// TIA Portal V17 export
// export: Created 2025-07-01T14:25:25.0430709Z, ExportSetting WithDefaults, DisplayName Totally Integrated Automation Portal, DisplayVersion V17 Update 8, DisplayName TIA Portal Openness, DisplayVersion V17 Update 8, DisplayName TIA Portal Version Control Interface, DisplayVersion V17, DisplayName SINAMICS Startdrive Advanced, DisplayVersion V17 SP2, DisplayName SINAMICS Startdrive G110M, G120, G120C, G120D, G120P, G115D, DisplayVersion V17 SP2, DisplayName SINAMICS Startdrive G130, G150, S120, S150, SINAMICS MV, S210, DisplayVersion V17 SP2, DisplayName STEP 7 Professional, DisplayVersion V17 Update 8, DisplayName SINUMERIK ONE STEP 7 Toolbox, DisplayVersion V17 Update 12, DisplayName SINUMERIK ONE PLC Basic Program Plus, DisplayVersion V17 Update 12, DisplayName SINUMERIK 840D sl STEP 7 Toolbox, DisplayVersion V17 Update 12, DisplayName STEP 7 Safety, DisplayVersion V17 Update 6, DisplayName WinCC Advanced, DisplayVersion V17 Update 8
FUNCTION_BLOCK "FB20202_TRUMPF_ACTIVE"   // FB20202, LAD
TITLE = FB20202 ACTIVE TRUMPF
{ S7_Optimized_Access := 'FALSE' }
VERSION : 0.1
// stored: AutoNumber false, IsIECCheckEnabled false, SetENOAutomatically false, UDAEnableTagReadback false
   VAR_INPUT
      iREADY_TO_EMISSION : Bool;
      "AIR COMPRESSED OK" : Bool;
      iPROGRAM_ACTIVE : Bool;
      iExternal_In : Bool;
      iMANUAL_START_REQUEST : Bool;
      iAUTO_START_REQUEST : Bool;
      iMANUAL_STOP_REQUEST : Bool;
      iAUTO_STOP_REQUEST : Bool;
      iProfile_Enable : Bool;
      iStart_Program_Request : Bool;
      iUNIT_RESET_LOCAL_SEQ : Bool;
      iSAFETY_GATES_CLOSED_LOCKED : Bool;
      iPART_PRESENTE : Bool;
      iLASER_READY_SC_STATUS : Bool;
      iMACHINE_ON_DELAYED : Bool;
      iZ_AXIS_IN_POSITION : Bool;
      iUNIT_NO : Int;
   END_VAR
   VAR_OUTPUT
      oEMISSION_SWITCH_ON : Bool;
      oPROGRAM_START : Bool;
      oALARM_PROGRAM_NOT_ACTIVE : Bool;
      oALARM_NO_LASER_EMISSION : Bool;
      oALARM_UNSAFE_STATE : Bool;
      oALARM_UNSAFE_AREA : Bool;
      "oALARM_LASER-DSS_ANALOG_MODE_MISMATCH" : Bool;
      oALARM_Z_AXIS_NOT_IN_POSITION : Bool;
      oSTATION_SEOC_ALARMS : Bool;
   END_VAR
   VAR DB_SPECIFIC
      DATA : "LASER ACTIVE";
      "TIMER FAULT 1" { S7_SetPoint := 'True'} : TON_TIME;
      "TIMER FAULT 2" { S7_SetPoint := 'True'} : TON_TIME;
      "DELAY EXTERNAL IN" { S7_SetPoint := 'True'} : TON_TIME;
   END_VAR
   VAR_TEMP
      DB_NUMBER : DInt;
   END_VAR
   VAR_TEMP   // added for the SCL form of the ladder/FBD networks
      _w1 : Bool;
   END_VAR
BEGIN

NETWORK
TITLE = READ INSTANCE DB NUMBER
      L     DINO;
      +     10#800000;
      T     #DB_NUMBER;

REGION Network 2: STOP GENERAL CONDITIONS
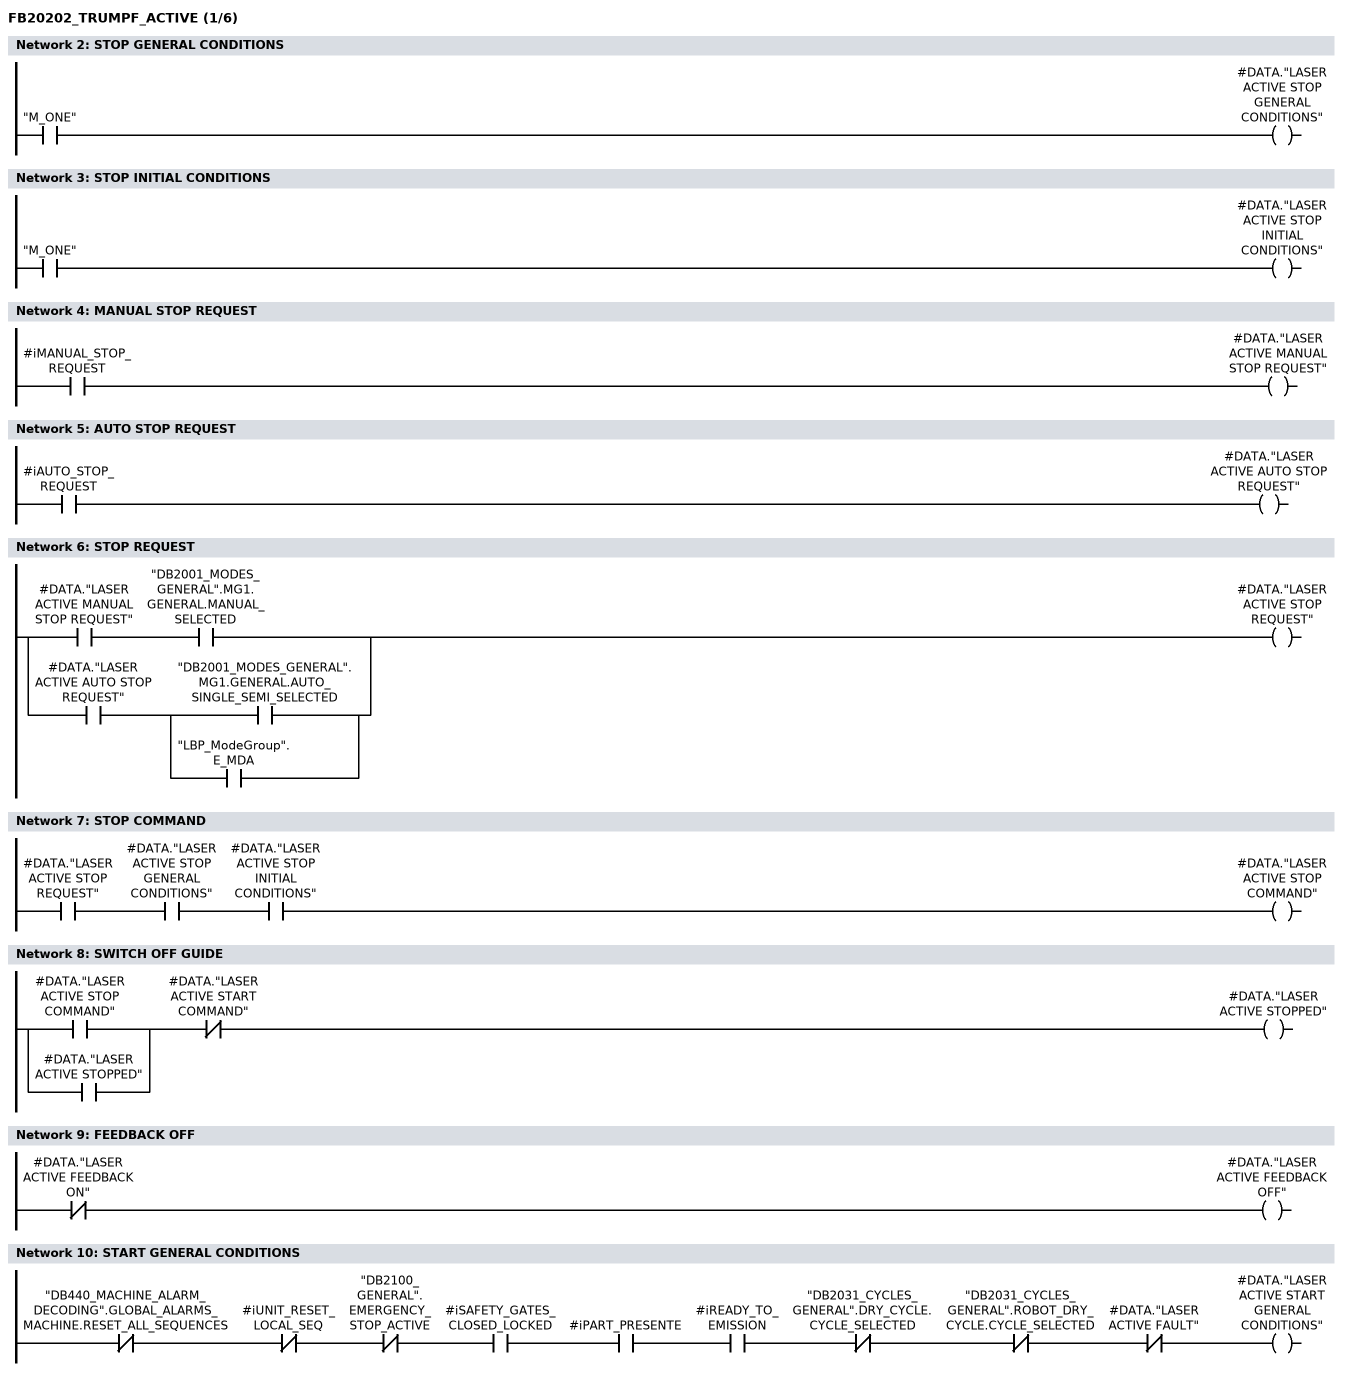
   RUNG wire#powerrail
      Contact( "M_ONE" )
      Coil( #DATA."LASER ACTIVE STOP GENERAL CONDITIONS" )
   END_RUNG
   // the same network as SCL:
   #DATA."LASER ACTIVE STOP GENERAL CONDITIONS" := "M_ONE";
END_REGION

REGION Network 3: STOP INITIAL CONDITIONS
   RUNG wire#powerrail
      Contact( "M_ONE" )
      Coil( #DATA."LASER ACTIVE STOP INITIAL CONDITIONS" )
   END_RUNG
   // the same network as SCL:
   #DATA."LASER ACTIVE STOP INITIAL CONDITIONS" := "M_ONE";
END_REGION

REGION Network 4: MANUAL STOP REQUEST
   RUNG wire#powerrail
      Contact( #iMANUAL_STOP_REQUEST )
      Coil( #DATA."LASER ACTIVE MANUAL STOP REQUEST" )
   END_RUNG
   // the same network as SCL:
   #DATA."LASER ACTIVE MANUAL STOP REQUEST" := #iMANUAL_STOP_REQUEST;
END_REGION

REGION Network 5: AUTO STOP REQUEST
   RUNG wire#powerrail
      Contact( #iAUTO_STOP_REQUEST )
      Coil( #DATA."LASER ACTIVE AUTO STOP REQUEST" )
   END_RUNG
   // the same network as SCL:
   #DATA."LASER ACTIVE AUTO STOP REQUEST" := #iAUTO_STOP_REQUEST;
END_REGION

REGION Network 6: STOP REQUEST
   RUNG wire#powerrail
      Contact( #DATA."LASER ACTIVE MANUAL STOP REQUEST" )
      Contact( "DB2001_MODES_GENERAL".MG1.GENERAL.MANUAL_SELECTED )
      wire#w1
      Coil( #DATA."LASER ACTIVE STOP REQUEST" )
   END_RUNG
   RUNG wire#powerrail
      Contact( #DATA."LASER ACTIVE AUTO STOP REQUEST" )
      wire#w2
      Contact( "DB2001_MODES_GENERAL".MG1.GENERAL.AUTO_SINGLE_SEMI_SELECTED )
   END_RUNG wire#w1
   RUNG wire#w2
      Contact( "LBP_ModeGroup".E_MDA )
   END_RUNG wire#w1
   // the same network as SCL:
   #DATA."LASER ACTIVE STOP REQUEST" := (#DATA."LASER ACTIVE MANUAL STOP REQUEST" AND "DB2001_MODES_GENERAL".MG1.GENERAL.MANUAL_SELECTED) OR (#DATA."LASER ACTIVE AUTO STOP REQUEST" AND ("DB2001_MODES_GENERAL".MG1.GENERAL.AUTO_SINGLE_SEMI_SELECTED OR "LBP_ModeGroup".E_MDA));
END_REGION

REGION Network 7: STOP COMMAND
   RUNG wire#powerrail
      Contact( #DATA."LASER ACTIVE STOP REQUEST" )
      Contact( #DATA."LASER ACTIVE STOP GENERAL CONDITIONS" )
      Contact( #DATA."LASER ACTIVE STOP INITIAL CONDITIONS" )
      Coil( #DATA."LASER ACTIVE STOP COMMAND" )
   END_RUNG
   // the same network as SCL:
   #DATA."LASER ACTIVE STOP COMMAND" := #DATA."LASER ACTIVE STOP REQUEST" AND #DATA."LASER ACTIVE STOP GENERAL CONDITIONS" AND #DATA."LASER ACTIVE STOP INITIAL CONDITIONS";
END_REGION

REGION Network 8: SWITCH OFF GUIDE
   RUNG wire#powerrail
      Contact( #DATA."LASER ACTIVE STOP COMMAND" )
      wire#w1
      I_Contact( #DATA."LASER ACTIVE START COMMAND" )
      Coil( #DATA."LASER ACTIVE STOPPED" )
   END_RUNG
   RUNG wire#powerrail
      Contact( #DATA."LASER ACTIVE STOPPED" )
   END_RUNG wire#w1
   // the same network as SCL:
   #DATA."LASER ACTIVE STOPPED" := (#DATA."LASER ACTIVE STOP COMMAND" OR #DATA."LASER ACTIVE STOPPED") AND NOT #DATA."LASER ACTIVE START COMMAND";
END_REGION

REGION Network 9: FEEDBACK OFF
   RUNG wire#powerrail
      I_Contact( #DATA."LASER ACTIVE FEEDBACK ON" )
      Coil( #DATA."LASER ACTIVE FEEDBACK OFF" )
   END_RUNG
   // the same network as SCL:
   #DATA."LASER ACTIVE FEEDBACK OFF" := NOT #DATA."LASER ACTIVE FEEDBACK ON";
END_REGION

REGION Network 10: START GENERAL CONDITIONS
   RUNG wire#powerrail
      I_Contact( "DB440_MACHINE_ALARM_DECODING".GLOBAL_ALARMS_MACHINE.RESET_ALL_SEQUENCES )
      I_Contact( #iUNIT_RESET_LOCAL_SEQ )
      I_Contact( "DB2100_GENERAL".EMERGENCY_STOP_ACTIVE )
      Contact( #iSAFETY_GATES_CLOSED_LOCKED )
      Contact( #iPART_PRESENTE )
      Contact( #iREADY_TO_EMISSION )
      I_Contact( "DB2031_CYCLES_GENERAL".DRY_CYCLE.CYCLE_SELECTED )
      I_Contact( "DB2031_CYCLES_GENERAL".ROBOT_DRY_CYCLE.CYCLE_SELECTED )
      I_Contact( #DATA."LASER ACTIVE FAULT" )
      Coil( #DATA."LASER ACTIVE START GENERAL CONDITIONS" )
   END_RUNG
   // the same network as SCL:
   #DATA."LASER ACTIVE START GENERAL CONDITIONS" := NOT "DB440_MACHINE_ALARM_DECODING".GLOBAL_ALARMS_MACHINE.RESET_ALL_SEQUENCES AND NOT #iUNIT_RESET_LOCAL_SEQ AND NOT "DB2100_GENERAL".EMERGENCY_STOP_ACTIVE AND #iSAFETY_GATES_CLOSED_LOCKED AND #iPART_PRESENTE AND #iREADY_TO_EMISSION AND NOT "DB2031_CYCLES_GENERAL".DRY_CYCLE.CYCLE_SELECTED AND NOT "DB2031_CYCLES_GENERAL".ROBOT_DRY_CYCLE.CYCLE_SELECTED AND NOT #DATA."LASER ACTIVE FAULT";
END_REGION

REGION Network 11: GENERAL CONDITIONS HELP
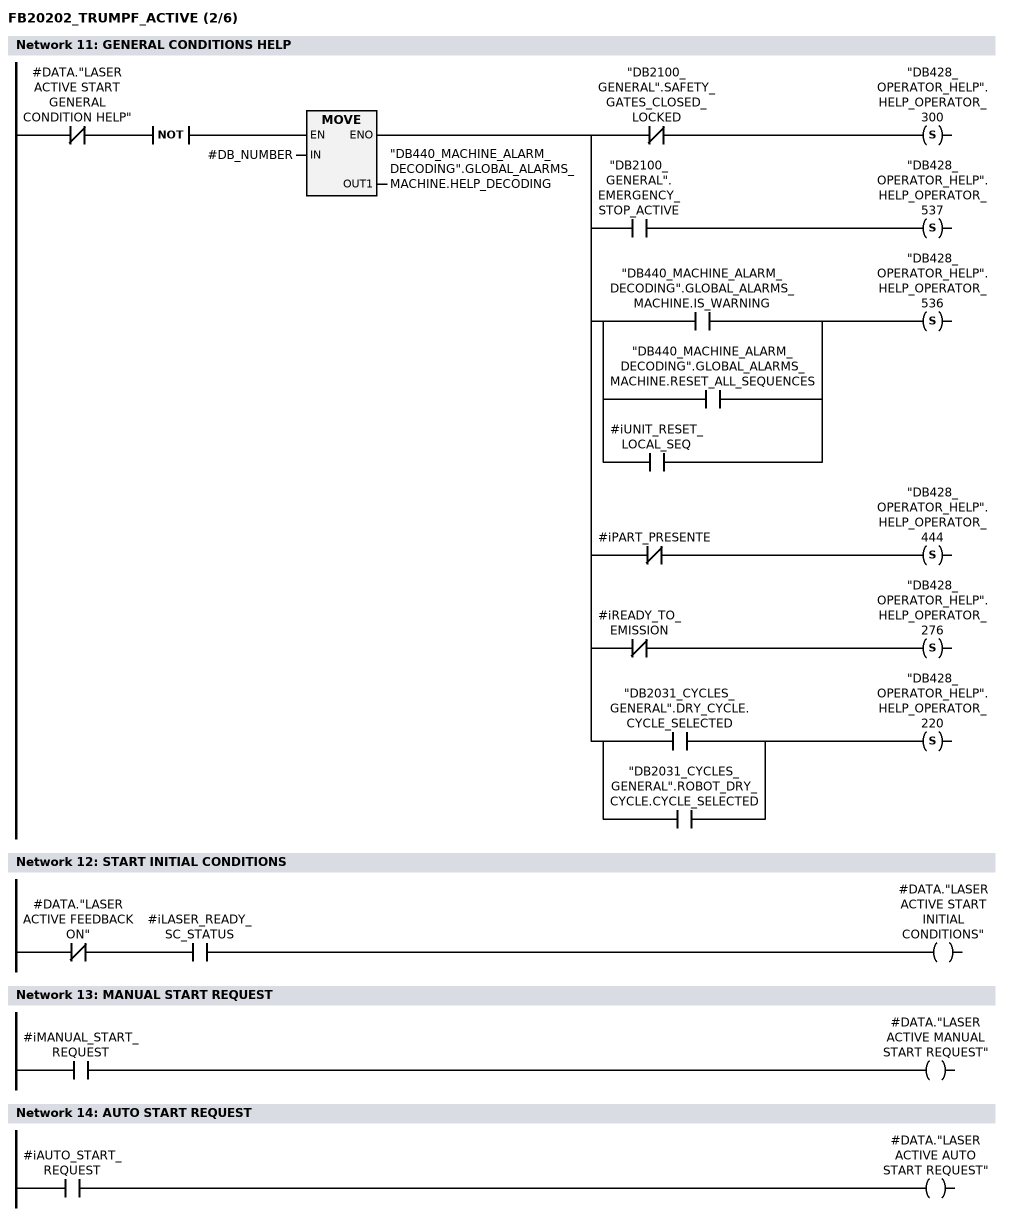
   RUNG wire#powerrail
      I_Contact( #DATA."LASER ACTIVE START GENERAL CONDITION HELP" )
      Not()
      Move(in := #DB_NUMBER, out1 => "DB440_MACHINE_ALARM_DECODING".GLOBAL_ALARMS_MACHINE.HELP_DECODING)
      wire#w1
      I_Contact( "DB2100_GENERAL".SAFETY_GATES_CLOSED_LOCKED )
      S_Coil( "DB428_OPERATOR_HELP".HELP_OPERATOR_300 )
   END_RUNG
   RUNG wire#w1
      Contact( "DB2100_GENERAL".EMERGENCY_STOP_ACTIVE )
      S_Coil( "DB428_OPERATOR_HELP".HELP_OPERATOR_537 )
   END_RUNG
   RUNG wire#w1
      Contact( "DB440_MACHINE_ALARM_DECODING".GLOBAL_ALARMS_MACHINE.IS_WARNING )
      wire#w2
      S_Coil( "DB428_OPERATOR_HELP".HELP_OPERATOR_536 )
   END_RUNG
   RUNG wire#w1
      Contact( "DB440_MACHINE_ALARM_DECODING".GLOBAL_ALARMS_MACHINE.RESET_ALL_SEQUENCES )
   END_RUNG wire#w2
   RUNG wire#w1
      Contact( #iUNIT_RESET_LOCAL_SEQ )
   END_RUNG wire#w2
   RUNG wire#w1
      I_Contact( #iPART_PRESENTE )
      S_Coil( "DB428_OPERATOR_HELP".HELP_OPERATOR_444 )
   END_RUNG
   RUNG wire#w1
      I_Contact( #iREADY_TO_EMISSION )
      S_Coil( "DB428_OPERATOR_HELP".HELP_OPERATOR_276 )
   END_RUNG
   RUNG wire#w1
      Contact( "DB2031_CYCLES_GENERAL".DRY_CYCLE.CYCLE_SELECTED )
      wire#w3
      S_Coil( "DB428_OPERATOR_HELP".HELP_OPERATOR_220 )
   END_RUNG
   RUNG wire#w1
      Contact( "DB2031_CYCLES_GENERAL".ROBOT_DRY_CYCLE.CYCLE_SELECTED )
   END_RUNG wire#w3
   // the same network as SCL:
   #_w1 := NOT (NOT #DATA."LASER ACTIVE START GENERAL CONDITION HELP");
   IF #_w1 THEN "DB440_MACHINE_ALARM_DECODING".GLOBAL_ALARMS_MACHINE.HELP_DECODING := #DB_NUMBER; END_IF;
   IF #_w1 AND NOT "DB2100_GENERAL".SAFETY_GATES_CLOSED_LOCKED THEN
       "DB428_OPERATOR_HELP".HELP_OPERATOR_300 := TRUE;
   END_IF;
   IF #_w1 AND "DB2100_GENERAL".EMERGENCY_STOP_ACTIVE THEN
       "DB428_OPERATOR_HELP".HELP_OPERATOR_537 := TRUE;
   END_IF;
   IF #_w1 AND ("DB440_MACHINE_ALARM_DECODING".GLOBAL_ALARMS_MACHINE.IS_WARNING OR "DB440_MACHINE_ALARM_DECODING".GLOBAL_ALARMS_MACHINE.RESET_ALL_SEQUENCES OR #iUNIT_RESET_LOCAL_SEQ) THEN
       "DB428_OPERATOR_HELP".HELP_OPERATOR_536 := TRUE;
   END_IF;
   IF #_w1 AND NOT #iPART_PRESENTE THEN "DB428_OPERATOR_HELP".HELP_OPERATOR_444 := TRUE; END_IF;
   IF #_w1 AND NOT #iREADY_TO_EMISSION THEN "DB428_OPERATOR_HELP".HELP_OPERATOR_276 := TRUE; END_IF;
   IF #_w1 AND ("DB2031_CYCLES_GENERAL".DRY_CYCLE.CYCLE_SELECTED OR "DB2031_CYCLES_GENERAL".ROBOT_DRY_CYCLE.CYCLE_SELECTED) THEN
       "DB428_OPERATOR_HELP".HELP_OPERATOR_220 := TRUE;
   END_IF;
END_REGION

REGION Network 12: START INITIAL CONDITIONS
   RUNG wire#powerrail
      I_Contact( #DATA."LASER ACTIVE FEEDBACK ON" )
      Contact( #iLASER_READY_SC_STATUS )
      Coil( #DATA."LASER ACTIVE START INITIAL CONDITIONS" )
   END_RUNG
   // the same network as SCL:
   #DATA."LASER ACTIVE START INITIAL CONDITIONS" := NOT #DATA."LASER ACTIVE FEEDBACK ON" AND #iLASER_READY_SC_STATUS;
END_REGION

REGION Network 13: MANUAL START REQUEST
   RUNG wire#powerrail
      Contact( #iMANUAL_START_REQUEST )
      Coil( #DATA."LASER ACTIVE MANUAL START REQUEST" )
   END_RUNG
   // the same network as SCL:
   #DATA."LASER ACTIVE MANUAL START REQUEST" := #iMANUAL_START_REQUEST;
END_REGION

REGION Network 14: AUTO START REQUEST
   RUNG wire#powerrail
      Contact( #iAUTO_START_REQUEST )
      Coil( #DATA."LASER ACTIVE AUTO START REQUEST" )
   END_RUNG
   // the same network as SCL:
   #DATA."LASER ACTIVE AUTO START REQUEST" := #iAUTO_START_REQUEST;
END_REGION

REGION Network 15: START REQUEST
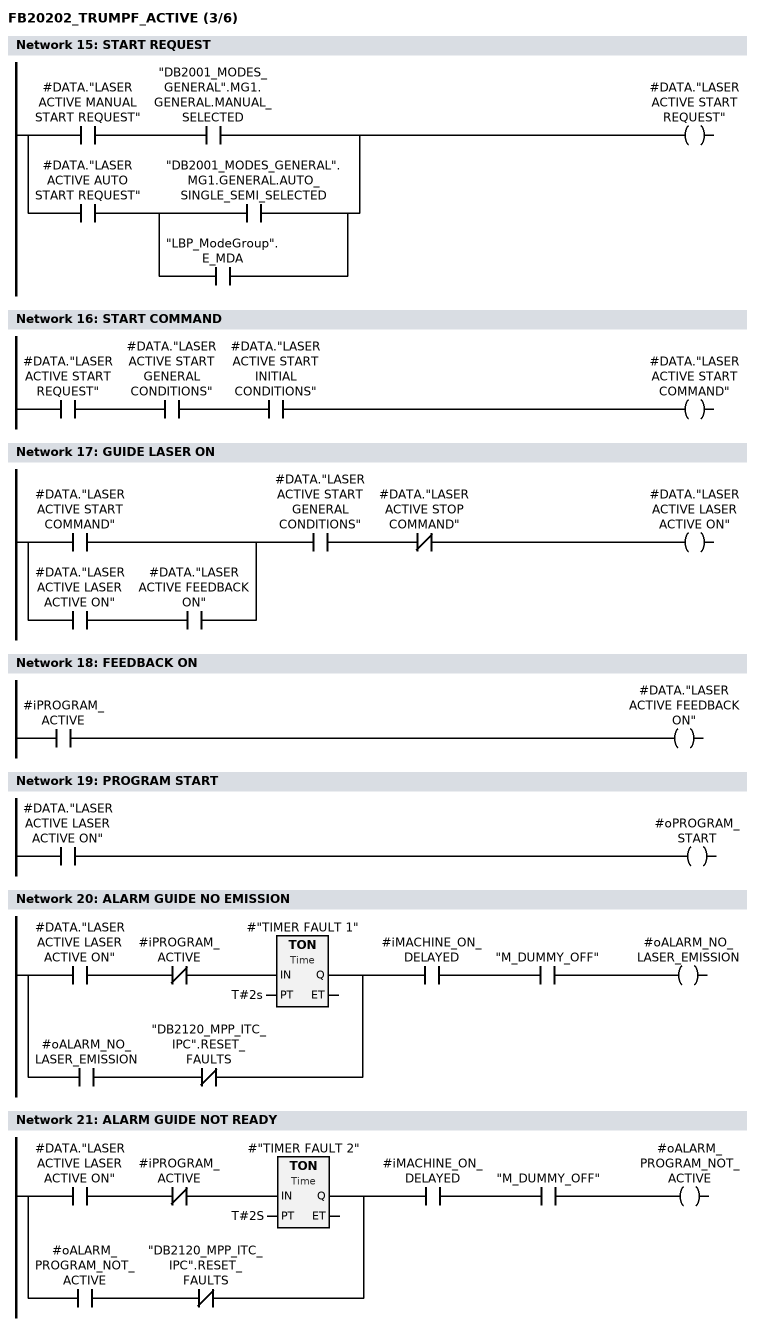
   RUNG wire#powerrail
      Contact( #DATA."LASER ACTIVE MANUAL START REQUEST" )
      Contact( "DB2001_MODES_GENERAL".MG1.GENERAL.MANUAL_SELECTED )
      wire#w1
      Coil( #DATA."LASER ACTIVE START REQUEST" )
   END_RUNG
   RUNG wire#powerrail
      Contact( #DATA."LASER ACTIVE AUTO START REQUEST" )
      wire#w2
      Contact( "DB2001_MODES_GENERAL".MG1.GENERAL.AUTO_SINGLE_SEMI_SELECTED )
   END_RUNG wire#w1
   RUNG wire#w2
      Contact( "LBP_ModeGroup".E_MDA )
   END_RUNG wire#w1
   // the same network as SCL:
   #DATA."LASER ACTIVE START REQUEST" := (#DATA."LASER ACTIVE MANUAL START REQUEST" AND "DB2001_MODES_GENERAL".MG1.GENERAL.MANUAL_SELECTED) OR (#DATA."LASER ACTIVE AUTO START REQUEST" AND ("DB2001_MODES_GENERAL".MG1.GENERAL.AUTO_SINGLE_SEMI_SELECTED OR "LBP_ModeGroup".E_MDA));
END_REGION

REGION Network 16: START COMMAND
   RUNG wire#powerrail
      Contact( #DATA."LASER ACTIVE START REQUEST" )
      Contact( #DATA."LASER ACTIVE START GENERAL CONDITIONS" )
      Contact( #DATA."LASER ACTIVE START INITIAL CONDITIONS" )
      Coil( #DATA."LASER ACTIVE START COMMAND" )
   END_RUNG
   // the same network as SCL:
   #DATA."LASER ACTIVE START COMMAND" := #DATA."LASER ACTIVE START REQUEST" AND #DATA."LASER ACTIVE START GENERAL CONDITIONS" AND #DATA."LASER ACTIVE START INITIAL CONDITIONS";
END_REGION

REGION Network 17: GUIDE LASER ON
   RUNG wire#powerrail
      Contact( #DATA."LASER ACTIVE START COMMAND" )
      wire#w1
      Contact( #DATA."LASER ACTIVE START GENERAL CONDITIONS" )
      I_Contact( #DATA."LASER ACTIVE STOP COMMAND" )
      Coil( #DATA."LASER ACTIVE LASER ACTIVE ON" )
   END_RUNG
   RUNG wire#powerrail
      Contact( #DATA."LASER ACTIVE LASER ACTIVE ON" )
      Contact( #DATA."LASER ACTIVE FEEDBACK ON" )
   END_RUNG wire#w1
   // the same network as SCL:
   #DATA."LASER ACTIVE LASER ACTIVE ON" := (#DATA."LASER ACTIVE START COMMAND" OR (#DATA."LASER ACTIVE LASER ACTIVE ON" AND #DATA."LASER ACTIVE FEEDBACK ON")) AND #DATA."LASER ACTIVE START GENERAL CONDITIONS" AND NOT #DATA."LASER ACTIVE STOP COMMAND";
END_REGION

REGION Network 18: FEEDBACK ON
   RUNG wire#powerrail
      Contact( #iPROGRAM_ACTIVE )
      Coil( #DATA."LASER ACTIVE FEEDBACK ON" )
   END_RUNG
   // the same network as SCL:
   #DATA."LASER ACTIVE FEEDBACK ON" := #iPROGRAM_ACTIVE;
END_REGION

REGION Network 19: PROGRAM START
   RUNG wire#powerrail
      Contact( #DATA."LASER ACTIVE LASER ACTIVE ON" )
      Coil( #oPROGRAM_START )
   END_RUNG
   // the same network as SCL:
   #oPROGRAM_START := #DATA."LASER ACTIVE LASER ACTIVE ON";
END_REGION

REGION Network 20: ALARM GUIDE NO EMISSION
   RUNG wire#powerrail
      Contact( #DATA."LASER ACTIVE LASER ACTIVE ON" )
      I_Contact( #iPROGRAM_ACTIVE )
      { S7_Templates := "time_type := Time" } #"TIMER FAULT 1".TON(pt := T#2s, et =>)
      wire#w1
      Contact( #iMACHINE_ON_DELAYED )
      Contact( "M_DUMMY_OFF" )
      Coil( #oALARM_NO_LASER_EMISSION )
   END_RUNG
   RUNG wire#powerrail
      Contact( #oALARM_NO_LASER_EMISSION )
      I_Contact( "DB2120_MPP_ITC_IPC".RESET_FAULTS )
   END_RUNG wire#w1
   // the same network as SCL:
   #"TIMER FAULT 1"(IN := #DATA."LASER ACTIVE LASER ACTIVE ON" AND NOT #iPROGRAM_ACTIVE, PT := T#2s);   // TON
   #oALARM_NO_LASER_EMISSION := (#"TIMER FAULT 1".Q OR (#oALARM_NO_LASER_EMISSION AND NOT "DB2120_MPP_ITC_IPC".RESET_FAULTS)) AND #iMACHINE_ON_DELAYED AND "M_DUMMY_OFF";
END_REGION

REGION Network 21: ALARM GUIDE NOT READY
   RUNG wire#powerrail
      Contact( #DATA."LASER ACTIVE LASER ACTIVE ON" )
      I_Contact( #iPROGRAM_ACTIVE )
      { S7_Templates := "time_type := Time" } #"TIMER FAULT 2".TON(pt := T#2S, et =>)
      wire#w1
      Contact( #iMACHINE_ON_DELAYED )
      Contact( "M_DUMMY_OFF" )
      Coil( #oALARM_PROGRAM_NOT_ACTIVE )
   END_RUNG
   RUNG wire#powerrail
      Contact( #oALARM_PROGRAM_NOT_ACTIVE )
      I_Contact( "DB2120_MPP_ITC_IPC".RESET_FAULTS )
   END_RUNG wire#w1
   // the same network as SCL:
   #"TIMER FAULT 2"(IN := #DATA."LASER ACTIVE LASER ACTIVE ON" AND NOT #iPROGRAM_ACTIVE, PT := T#2S);   // TON
   #oALARM_PROGRAM_NOT_ACTIVE := (#"TIMER FAULT 2".Q OR (#oALARM_PROGRAM_NOT_ACTIVE AND NOT "DB2120_MPP_ITC_IPC".RESET_FAULTS)) AND #iMACHINE_ON_DELAYED AND "M_DUMMY_OFF";
END_REGION

REGION Network 22: ALARM GUIDE NOT READY
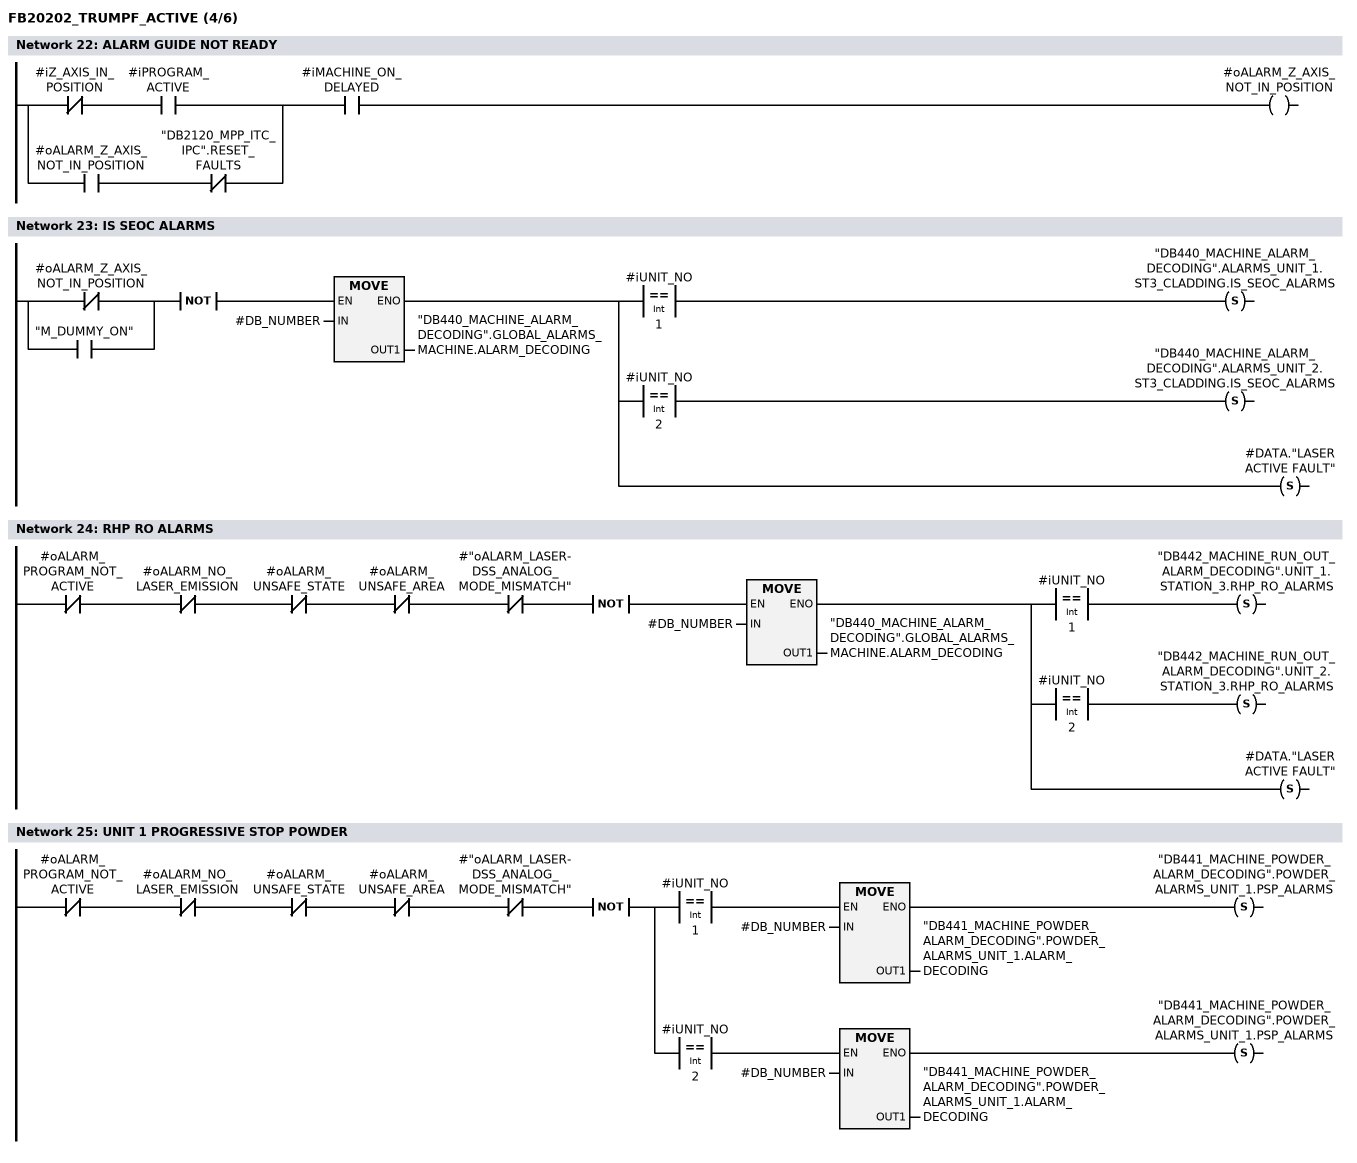
   RUNG wire#powerrail
      I_Contact( #iZ_AXIS_IN_POSITION )
      Contact( #iPROGRAM_ACTIVE )
      wire#w1
      Contact( #iMACHINE_ON_DELAYED )
      Coil( #oALARM_Z_AXIS_NOT_IN_POSITION )
   END_RUNG
   RUNG wire#powerrail
      Contact( #oALARM_Z_AXIS_NOT_IN_POSITION )
      I_Contact( "DB2120_MPP_ITC_IPC".RESET_FAULTS )
   END_RUNG wire#w1
   // the same network as SCL:
   #oALARM_Z_AXIS_NOT_IN_POSITION := ((NOT #iZ_AXIS_IN_POSITION AND #iPROGRAM_ACTIVE) OR (#oALARM_Z_AXIS_NOT_IN_POSITION AND NOT "DB2120_MPP_ITC_IPC".RESET_FAULTS)) AND #iMACHINE_ON_DELAYED;
END_REGION

REGION Network 23: IS SEOC ALARMS
   RUNG wire#powerrail
      I_Contact( #oALARM_Z_AXIS_NOT_IN_POSITION )
      wire#w1
      Not()
      Move(in := #DB_NUMBER, out1 => "DB440_MACHINE_ALARM_DECODING".GLOBAL_ALARMS_MACHINE.ALARM_DECODING)
      wire#w2
      { S7_Templates := "SrcType := Int" } EQ_Contact(in1 := #iUNIT_NO, in2 := 1)
      S_Coil( "DB440_MACHINE_ALARM_DECODING".ALARMS_UNIT_1.ST3_CLADDING.IS_SEOC_ALARMS )
   END_RUNG
   RUNG wire#powerrail
      Contact( "M_DUMMY_ON" )
   END_RUNG wire#w1
   RUNG wire#w2
      { S7_Templates := "SrcType := Int" } EQ_Contact(in1 := #iUNIT_NO, in2 := 2)
      S_Coil( "DB440_MACHINE_ALARM_DECODING".ALARMS_UNIT_2.ST3_CLADDING.IS_SEOC_ALARMS )
   END_RUNG
   RUNG wire#w2
      S_Coil( #DATA."LASER ACTIVE FAULT" )
   END_RUNG
   // the same network as SCL:
   #_w1 := NOT (NOT #oALARM_Z_AXIS_NOT_IN_POSITION OR "M_DUMMY_ON");
   IF #_w1 THEN "DB440_MACHINE_ALARM_DECODING".GLOBAL_ALARMS_MACHINE.ALARM_DECODING := #DB_NUMBER; END_IF;
   IF #_w1 AND (#iUNIT_NO = 1) THEN
       "DB440_MACHINE_ALARM_DECODING".ALARMS_UNIT_1.ST3_CLADDING.IS_SEOC_ALARMS := TRUE;
   END_IF;
   IF #_w1 AND (#iUNIT_NO = 2) THEN
       "DB440_MACHINE_ALARM_DECODING".ALARMS_UNIT_2.ST3_CLADDING.IS_SEOC_ALARMS := TRUE;
   END_IF;
   IF #_w1 THEN #DATA."LASER ACTIVE FAULT" := TRUE; END_IF;
END_REGION

REGION Network 24: RHP RO ALARMS
   RUNG wire#powerrail
      I_Contact( #oALARM_PROGRAM_NOT_ACTIVE )
      I_Contact( #oALARM_NO_LASER_EMISSION )
      I_Contact( #oALARM_UNSAFE_STATE )
      I_Contact( #oALARM_UNSAFE_AREA )
      I_Contact( #"oALARM_LASER-DSS_ANALOG_MODE_MISMATCH" )
      Not()
      Move(in := #DB_NUMBER, out1 => "DB440_MACHINE_ALARM_DECODING".GLOBAL_ALARMS_MACHINE.ALARM_DECODING)
      wire#w1
      { S7_Templates := "SrcType := Int" } EQ_Contact(in1 := #iUNIT_NO, in2 := 1)
      S_Coil( "DB442_MACHINE_RUN_OUT_ALARM_DECODING".UNIT_1.STATION_3.RHP_RO_ALARMS )
   END_RUNG
   RUNG wire#w1
      { S7_Templates := "SrcType := Int" } EQ_Contact(in1 := #iUNIT_NO, in2 := 2)
      S_Coil( "DB442_MACHINE_RUN_OUT_ALARM_DECODING".UNIT_2.STATION_3.RHP_RO_ALARMS )
   END_RUNG
   RUNG wire#w1
      S_Coil( #DATA."LASER ACTIVE FAULT" )
   END_RUNG
   // the same network as SCL:
   #_w1 := NOT (NOT #oALARM_PROGRAM_NOT_ACTIVE AND NOT #oALARM_NO_LASER_EMISSION AND NOT #oALARM_UNSAFE_STATE AND NOT #oALARM_UNSAFE_AREA AND NOT #"oALARM_LASER-DSS_ANALOG_MODE_MISMATCH");
   IF #_w1 THEN "DB440_MACHINE_ALARM_DECODING".GLOBAL_ALARMS_MACHINE.ALARM_DECODING := #DB_NUMBER; END_IF;
   IF #_w1 AND (#iUNIT_NO = 1) THEN
       "DB442_MACHINE_RUN_OUT_ALARM_DECODING".UNIT_1.STATION_3.RHP_RO_ALARMS := TRUE;
   END_IF;
   IF #_w1 AND (#iUNIT_NO = 2) THEN
       "DB442_MACHINE_RUN_OUT_ALARM_DECODING".UNIT_2.STATION_3.RHP_RO_ALARMS := TRUE;
   END_IF;
   IF #_w1 THEN #DATA."LASER ACTIVE FAULT" := TRUE; END_IF;
END_REGION

REGION Network 25: UNIT 1 PROGRESSIVE STOP POWDER
   RUNG wire#powerrail
      I_Contact( #oALARM_PROGRAM_NOT_ACTIVE )
      I_Contact( #oALARM_NO_LASER_EMISSION )
      I_Contact( #oALARM_UNSAFE_STATE )
      I_Contact( #oALARM_UNSAFE_AREA )
      I_Contact( #"oALARM_LASER-DSS_ANALOG_MODE_MISMATCH" )
      Not()
      wire#w1
      { S7_Templates := "SrcType := Int" } EQ_Contact(in1 := #iUNIT_NO, in2 := 1)
      Move(in := #DB_NUMBER, out1 => "DB441_MACHINE_POWDER_ALARM_DECODING".POWDER_ALARMS_UNIT_1.ALARM_DECODING)
      S_Coil( "DB441_MACHINE_POWDER_ALARM_DECODING".POWDER_ALARMS_UNIT_1.PSP_ALARMS )
   END_RUNG
   RUNG wire#w1
      { S7_Templates := "SrcType := Int" } EQ_Contact(in1 := #iUNIT_NO, in2 := 2)
      Move(in := #DB_NUMBER, out1 => "DB441_MACHINE_POWDER_ALARM_DECODING".POWDER_ALARMS_UNIT_1.ALARM_DECODING)
      S_Coil( "DB441_MACHINE_POWDER_ALARM_DECODING".POWDER_ALARMS_UNIT_1.PSP_ALARMS )
   END_RUNG
   // the same network as SCL:
   #_w1 := NOT (NOT #oALARM_PROGRAM_NOT_ACTIVE AND NOT #oALARM_NO_LASER_EMISSION AND NOT #oALARM_UNSAFE_STATE AND NOT #oALARM_UNSAFE_AREA AND NOT #"oALARM_LASER-DSS_ANALOG_MODE_MISMATCH");
   IF #_w1 AND (#iUNIT_NO = 1) THEN
       "DB441_MACHINE_POWDER_ALARM_DECODING".POWDER_ALARMS_UNIT_1.ALARM_DECODING := #DB_NUMBER;
       "DB441_MACHINE_POWDER_ALARM_DECODING".POWDER_ALARMS_UNIT_1.PSP_ALARMS := TRUE;
   END_IF;
   IF #_w1 AND (#iUNIT_NO = 2) THEN
       "DB441_MACHINE_POWDER_ALARM_DECODING".POWDER_ALARMS_UNIT_1.ALARM_DECODING := #DB_NUMBER;
       "DB441_MACHINE_POWDER_ALARM_DECODING".POWDER_ALARMS_UNIT_1.PSP_ALARMS := TRUE;
   END_IF;
END_REGION

REGION Network 26: UNIT 2 MAINTAIN POWDER
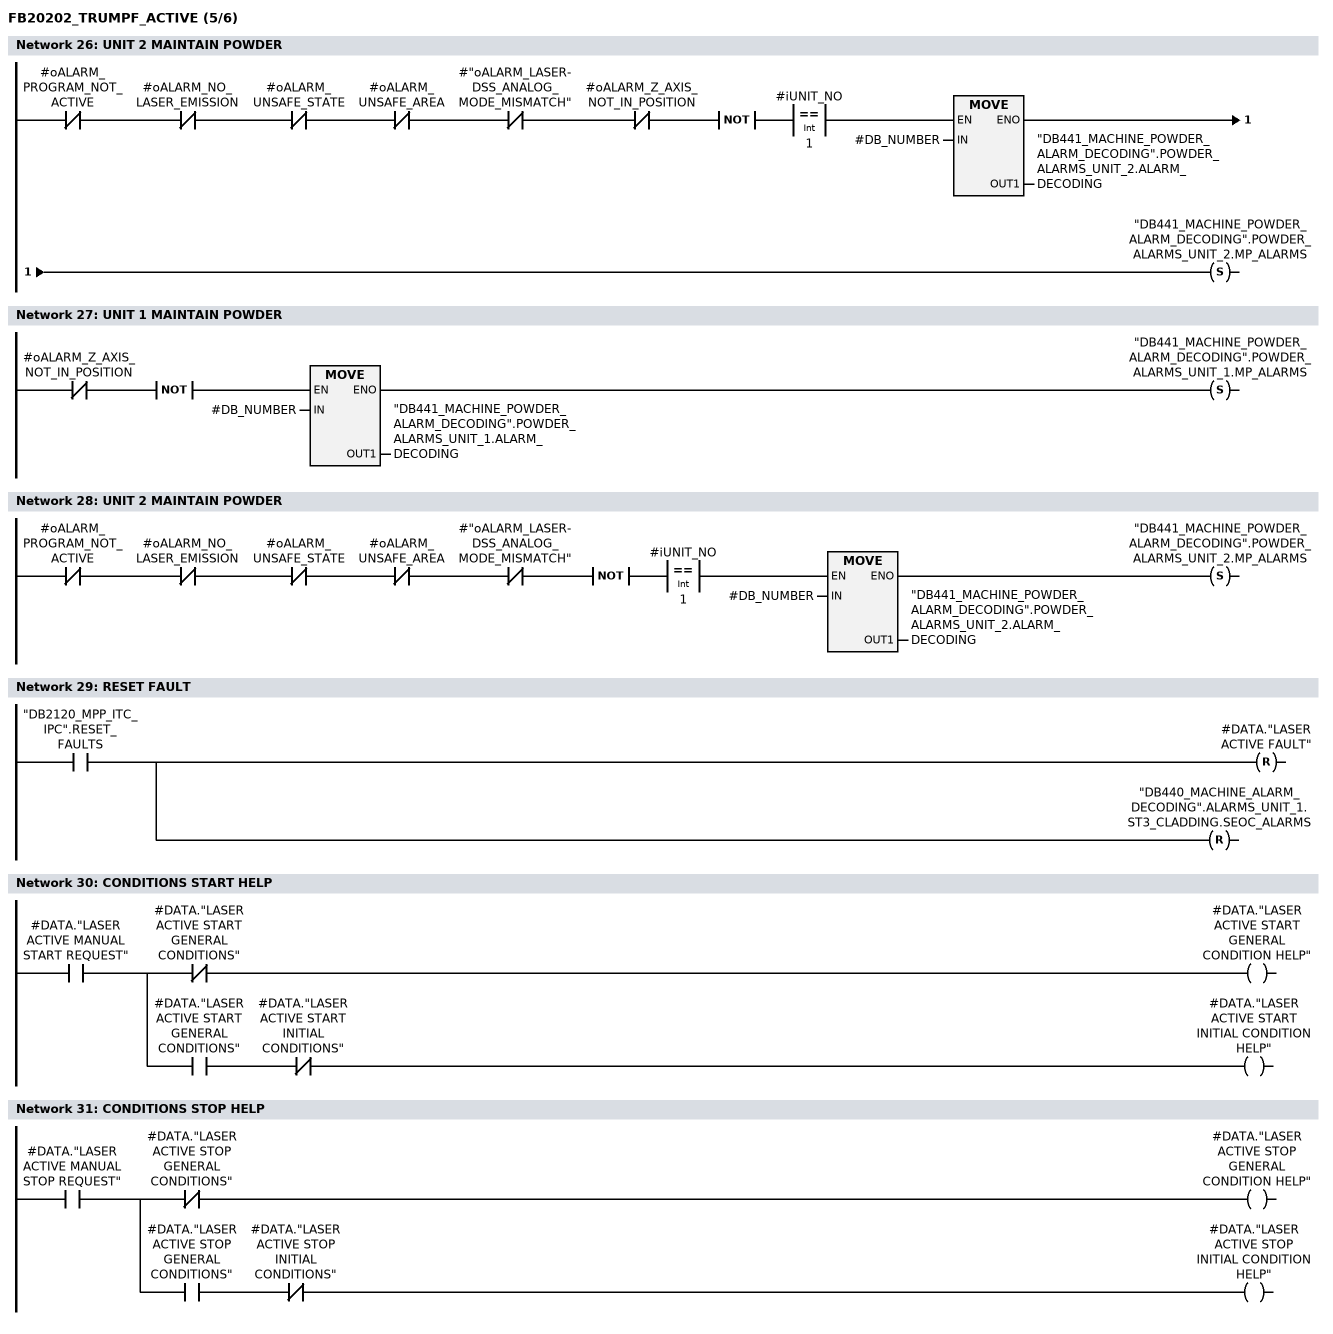
   RUNG wire#powerrail
      I_Contact( #oALARM_PROGRAM_NOT_ACTIVE )
      I_Contact( #oALARM_NO_LASER_EMISSION )
      I_Contact( #oALARM_UNSAFE_STATE )
      I_Contact( #oALARM_UNSAFE_AREA )
      I_Contact( #"oALARM_LASER-DSS_ANALOG_MODE_MISMATCH" )
      I_Contact( #oALARM_Z_AXIS_NOT_IN_POSITION )
      Not()
      { S7_Templates := "SrcType := Int" } EQ_Contact(in1 := #iUNIT_NO, in2 := 1)
      Move(in := #DB_NUMBER, out1 => "DB441_MACHINE_POWDER_ALARM_DECODING".POWDER_ALARMS_UNIT_2.ALARM_DECODING)
      S_Coil( "DB441_MACHINE_POWDER_ALARM_DECODING".POWDER_ALARMS_UNIT_2.MP_ALARMS )
   END_RUNG
   // the same network as SCL:
   IF NOT (NOT #oALARM_PROGRAM_NOT_ACTIVE AND NOT #oALARM_NO_LASER_EMISSION AND NOT #oALARM_UNSAFE_STATE AND NOT #oALARM_UNSAFE_AREA AND NOT #"oALARM_LASER-DSS_ANALOG_MODE_MISMATCH" AND NOT #oALARM_Z_AXIS_NOT_IN_POSITION) AND (#iUNIT_NO = 1) THEN
       "DB441_MACHINE_POWDER_ALARM_DECODING".POWDER_ALARMS_UNIT_2.ALARM_DECODING := #DB_NUMBER;
       "DB441_MACHINE_POWDER_ALARM_DECODING".POWDER_ALARMS_UNIT_2.MP_ALARMS := TRUE;
   END_IF;
END_REGION

REGION Network 27: UNIT 1 MAINTAIN POWDER
   RUNG wire#powerrail
      I_Contact( #oALARM_Z_AXIS_NOT_IN_POSITION )
      Not()
      Move(in := #DB_NUMBER, out1 => "DB441_MACHINE_POWDER_ALARM_DECODING".POWDER_ALARMS_UNIT_1.ALARM_DECODING)
      S_Coil( "DB441_MACHINE_POWDER_ALARM_DECODING".POWDER_ALARMS_UNIT_1.MP_ALARMS )
   END_RUNG
   // the same network as SCL:
   IF NOT (NOT #oALARM_Z_AXIS_NOT_IN_POSITION) THEN
       "DB441_MACHINE_POWDER_ALARM_DECODING".POWDER_ALARMS_UNIT_1.ALARM_DECODING := #DB_NUMBER;
       "DB441_MACHINE_POWDER_ALARM_DECODING".POWDER_ALARMS_UNIT_1.MP_ALARMS := TRUE;
   END_IF;
END_REGION

REGION Network 28: UNIT 2 MAINTAIN POWDER
   RUNG wire#powerrail
      I_Contact( #oALARM_PROGRAM_NOT_ACTIVE )
      I_Contact( #oALARM_NO_LASER_EMISSION )
      I_Contact( #oALARM_UNSAFE_STATE )
      I_Contact( #oALARM_UNSAFE_AREA )
      I_Contact( #"oALARM_LASER-DSS_ANALOG_MODE_MISMATCH" )
      Not()
      { S7_Templates := "SrcType := Int" } EQ_Contact(in1 := #iUNIT_NO, in2 := 1)
      Move(in := #DB_NUMBER, out1 => "DB441_MACHINE_POWDER_ALARM_DECODING".POWDER_ALARMS_UNIT_2.ALARM_DECODING)
      S_Coil( "DB441_MACHINE_POWDER_ALARM_DECODING".POWDER_ALARMS_UNIT_2.MP_ALARMS )
   END_RUNG
   // the same network as SCL:
   IF NOT (NOT #oALARM_PROGRAM_NOT_ACTIVE AND NOT #oALARM_NO_LASER_EMISSION AND NOT #oALARM_UNSAFE_STATE AND NOT #oALARM_UNSAFE_AREA AND NOT #"oALARM_LASER-DSS_ANALOG_MODE_MISMATCH") AND (#iUNIT_NO = 1) THEN
       "DB441_MACHINE_POWDER_ALARM_DECODING".POWDER_ALARMS_UNIT_2.ALARM_DECODING := #DB_NUMBER;
       "DB441_MACHINE_POWDER_ALARM_DECODING".POWDER_ALARMS_UNIT_2.MP_ALARMS := TRUE;
   END_IF;
END_REGION

REGION Network 29: RESET FAULT
   RUNG wire#powerrail
      Contact( "DB2120_MPP_ITC_IPC".RESET_FAULTS )
      wire#w1
      R_Coil( #DATA."LASER ACTIVE FAULT" )
   END_RUNG
   RUNG wire#w1
      R_Coil( "DB440_MACHINE_ALARM_DECODING".ALARMS_UNIT_1.ST3_CLADDING.SEOC_ALARMS )
   END_RUNG
   // the same network as SCL:
   IF "DB2120_MPP_ITC_IPC".RESET_FAULTS THEN
       #DATA."LASER ACTIVE FAULT" := FALSE;
       "DB440_MACHINE_ALARM_DECODING".ALARMS_UNIT_1.ST3_CLADDING.SEOC_ALARMS := FALSE;
   END_IF;
END_REGION

REGION Network 30: CONDITIONS START HELP
   RUNG wire#powerrail
      Contact( #DATA."LASER ACTIVE MANUAL START REQUEST" )
      wire#w1
      I_Contact( #DATA."LASER ACTIVE START GENERAL CONDITIONS" )
      Coil( #DATA."LASER ACTIVE START GENERAL CONDITION HELP" )
   END_RUNG
   RUNG wire#w1
      Contact( #DATA."LASER ACTIVE START GENERAL CONDITIONS" )
      I_Contact( #DATA."LASER ACTIVE START INITIAL CONDITIONS" )
      Coil( #DATA."LASER ACTIVE START INITIAL CONDITION HELP" )
   END_RUNG
   // the same network as SCL:
   #DATA."LASER ACTIVE START GENERAL CONDITION HELP" := #DATA."LASER ACTIVE MANUAL START REQUEST" AND NOT #DATA."LASER ACTIVE START GENERAL CONDITIONS";
   #DATA."LASER ACTIVE START INITIAL CONDITION HELP" := #DATA."LASER ACTIVE MANUAL START REQUEST" AND #DATA."LASER ACTIVE START GENERAL CONDITIONS" AND NOT #DATA."LASER ACTIVE START INITIAL CONDITIONS";
END_REGION

REGION Network 31: CONDITIONS STOP HELP
   RUNG wire#powerrail
      Contact( #DATA."LASER ACTIVE MANUAL STOP REQUEST" )
      wire#w1
      I_Contact( #DATA."LASER ACTIVE STOP GENERAL CONDITIONS" )
      Coil( #DATA."LASER ACTIVE STOP GENERAL CONDITION HELP" )
   END_RUNG
   RUNG wire#w1
      Contact( #DATA."LASER ACTIVE STOP GENERAL CONDITIONS" )
      I_Contact( #DATA."LASER ACTIVE STOP INITIAL CONDITIONS" )
      Coil( #DATA."LASER ACTIVE STOP INITIAL CONDITION HELP" )
   END_RUNG
   // the same network as SCL:
   #DATA."LASER ACTIVE STOP GENERAL CONDITION HELP" := #DATA."LASER ACTIVE MANUAL STOP REQUEST" AND NOT #DATA."LASER ACTIVE STOP GENERAL CONDITIONS";
   #DATA."LASER ACTIVE STOP INITIAL CONDITION HELP" := #DATA."LASER ACTIVE MANUAL STOP REQUEST" AND #DATA."LASER ACTIVE STOP GENERAL CONDITIONS" AND NOT #DATA."LASER ACTIVE STOP INITIAL CONDITIONS";
END_REGION

REGION Network 32: SWITCH ON OUTPUT GUIDE LASER
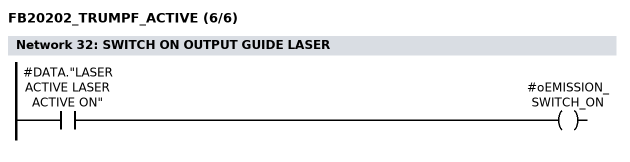
   RUNG wire#powerrail
      Contact( #DATA."LASER ACTIVE LASER ACTIVE ON" )
      Coil( #oEMISSION_SWITCH_ON )
   END_RUNG
   // the same network as SCL:
   #oEMISSION_SWITCH_ON := #DATA."LASER ACTIVE LASER ACTIVE ON";
END_REGION
END_FUNCTION_BLOCK
